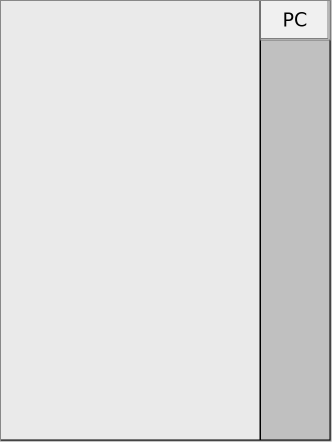
VISUALIZATION V_Main_Mob  // 332x442
    Rectangle (260,0 70x440)
    Rectangle (0,0 260x440)
    Button (260,0 70x40), "PC"
        OnMouseUp: change screen: V_Main_PC
END_VISUALIZATION

(* stored: Version 1.1.0.1, ProductVersion 3.1.4018.5
   Visu V_Main_Mob: Id {fd384381-eeb9-4b40-adba-8ee6951362c1} *)
